PROGRAM MAIN
VAR
	nC: INT;
	nC2: INT;
	nC3: INT;
	nC4: INT;
END_VAR

nC:=nC+1;
nC2:=nC2+1;
nC3:=nC3+1;
nC4:=nC4+1;

END_PROGRAM

(* stored: Version 1.1.0.1
   POU MAIN: Id {ffeaeec1-8acb-4087-8b37-b8c98acc680d}, SpecialFunc None *)
